FUNCTION F_CalcTD20Checksum : BYTE
VAR_INPUT
    i_abData: ARRAY[0..23] OF BYTE;
END_VAR
VAR
    bChecksum: BYTE;
    i: INT;
END_VAR

bChecksum := i_abData[0];
FOR i:=1 TO 22 DO
    bChecksum := bChecksum XOR i_abData[i];
END_FOR
F_CalcTD20Checksum := bChecksum;

END_FUNCTION

(* stored: Version 1.1.0.1
   POU F_CalcTD20Checksum: Id {59d21b56-e4d7-4723-a1de-95977cb48cdd}, SpecialFunc None *)
